(* PLC project Unnamed, Неизвестно Unnamed 1 *)
(* stored: creationDateTime 2024-03-27T15:49:36, modificationDateTime 2024-03-27T16:20:57 *)

PROGRAM PWM
  VAR
    LocalVar0 : DINT;
    LocalVar1 : DINT;
  END_VAR

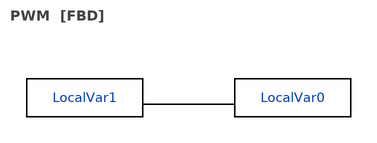
(* FBD diagram, written out as Structured Text *)
LocalVar0 := LocalVar1;
END_PROGRAM

CONFIGURATION Config0
  RESOURCE Res0 ON PLC
    TASK task0(INTERVAL := T#20ms, PRIORITY := 0);
    PROGRAM instance0 WITH task0 : PWM;
  END_RESOURCE
END_CONFIGURATION
